FUNCTION_BLOCK MockError EXTENDS Error
VAR
	_errorType : T_MAXSTRING;
	_message : T_MAXSTRING;
END_VAR

PROPERTY PUBLIC ErrorType : T_MAXSTRING
GET
ErrorType := _errorType;
END_GET
END_PROPERTY

METHOD FB_init : BOOL
VAR_INPUT
	bInitRetains : BOOL; // if TRUE, the retain variables are initialized (warm start / cold start)
	bInCopyCode : BOOL;  // if TRUE, the instance afterwards gets moved into the copy code (online change)
	MockErrorType : T_MAXSTRING;
	MockMessage : T_MAXSTRING;
END_VAR
_errorType := MockErrorType;
_message := MockMessage;
END_METHOD

PROPERTY PUBLIC Message : T_MAXSTRING
GET
Message := _message;
END_GET
END_PROPERTY

END_FUNCTION_BLOCK

(* stored: Version 1.1.0.1, ProductVersion 3.1.4024.12
   POU MockError: Id {94603a1c-dc28-48c9-8694-3e72a05d220a}, SpecialFunc None
   Folder Constructor: Id {27b801fc-bbe0-46d6-938e-57bd1586bd9f}
   Property ErrorType: Id {b31af701-52ea-4420-9792-9c7db4e64b06}
   Get Get: Id {06c2f282-1262-4919-bbcf-b1af7bc7609d}
   Method FB_init: Id {a4bb2593-4914-4b71-8fc6-6f81a2353213}
   Property Message: Id {d3821f36-8a34-4c76-a838-c356d8886767}
   Get Get: Id {2f07bf9b-9413-47ee-b5ba-6c49beef0cfc} *)
